Yaskawa INFORM job: SBTOPEN.JBI

/JOB
//NAME SBTOPEN
//POS
///NPOS 0,0,0,0,0,0
//INST
///DATE 2020/09/26 16:06
///ATTR SC,RW,MC
///GROUP1 RB1
///LVARS 0,1,1,0,1,0,0,0
NOP
GETARG LS000 IARG#(1)
GETARG LD000 IARG#(2)
GETARG LI000 IARG#(3)
SET S070 LS000
SET D070 LD000
SET I010 LI000
SET B069 0
SKILLSND "SpeedbotClose"
SKILLSND "SpeedbotOpen"
WAIT B069=1 T=I010
end
